// TIA Portal V16 export
// export: Created 2024-04-26T21:24:43.2623073Z, ExportSetting WithDefaults, DisplayName Totally Integrated Automation Portal, DisplayVersion V16, DisplayName TIA Portal Version Control Interface, DisplayVersion V16, DisplayName TIA Portal Openness, DisplayVersion V16, DisplayName STEP 7 Professional, DisplayVersion V16, DisplayName STEP 7 Safety, DisplayVersion V16, DisplayName WinCC Professional, DisplayVersion V16
DATA_BLOCK "MC_MoveRelative_DB_3"   // DB19
// stored: AutoNumber true, InstanceOfName MC_MoveRelative, OfSystemLibElement MC_MoveRelative, OfSystemLibVersion 6.0
"MC_MoveRelative"
   // VAR_INPUT
   //    Axis : TO_PositioningAxis;
   //    Execute : Bool;
   //    Distance : Real;
   //    Velocity : Real;
   // END_VAR
   // VAR_OUTPUT
   //    Done : Bool;
   //    Busy : Bool;
   //    CommandAborted : Bool;
   //    Error : Bool;
   //    ErrorID : Word;
   //    ErrorInfo : Word;
   // END_VAR
   // VAR
   //    FB_ID : DInt;
   // END_VAR
BEGIN
END_DATA_BLOCK
